FUNCTION_BLOCK Updater_1 IMPLEMENTS ITF_Updater
VAR CONSTANT
    PacketID  				: BYTE := 1;
    PacketVersion 			: BYTE := 1;
	PacketSize				: BYTE := 66;
END_VAR
VAR
	TempBuffer				: ARRAY [0..PacketSize - 1] OF BYTE;	

	ApplyOkCount            : UDINT;
    ApplyLengthErrorCount   : UDINT;
    ApplyBufferTooSmall     : UDINT;
END_VAR

METHOD GetTypeID : BYTE
GetTypeID := PacketID;
END_METHOD

METHOD GetVersion : BYTE
GetVersion := PacketVersion;
END_METHOD

METHOD TryApplyPayload : HRESULT
VAR_INPUT
	PacketAddress	: PVOID;
	PacketLength	: UINT;
	EspHost			: ITF_EspHost;
END_VAR
VAR
    BufferAddress : PVOID;
    BufferSize    : UDINT;
END_VAR
TryApplyPayload := S_PENDING;

IF PacketLength <> PacketSize THEN
	
    ApplyLengthErrorCount := ApplyLengthErrorCount + 1;
	
	TryApplyPayload := -1;
	
	RETURN;
	
END_IF

IF NOT EspHost.GetDataBuffer(BufferAddress, BufferSize) THEN
	
	TryApplyPayload := -2;

    RETURN;
	
END_IF

IF PacketLength > BufferSize THEN
	
    ApplyBufferTooSmall := ApplyBufferTooSmall + 1;
	
    TryApplyPayload := -3;
    
	RETURN;

END_IF



MEMCPY(BufferAddress, PacketAddress, PacketLength);

ApplyOkCount := ApplyOkCount + 1;

TryApplyPayload := S_OK;          // success

RETURN;
END_METHOD

METHOD TryGetContents : HRESULT
VAR_INPUT
	Host	: ITF_EspHost;
	Content	: REFERENCE TO STRING(1024);
END_VAR
VAR
    BufferAddress 	: PVOID;
    BufferSize   	: UDINT;
	td9 			: ULINT;
END_VAR
TryGetContents := S_PENDING;

Content := '{"Error" : "No_Data_Available"}';

IF NOT Host.GetDataBuffer(BufferAddress, BufferSize) THEN

	TryGetContents := -1;	

    RETURN;
	
END_IF

IF MEMCPY(ADR(TempBuffer), BufferAddress, BufferSize) <= 0 THEN
	
	TryGetContents := -2;
	
	RETURN;

END_IF

Content := '';

Content := CONCAT(Content, '{"Test_Data_1" : ');
Content := CONCAT(Content, TO_STRING(TempBuffer[48]));
Content := CONCAT(Content, ', "Test_Data_2" : ');
Content := CONCAT(Content, TO_STRING(TempBuffer[49]));
Content := CONCAT(Content, ', "Test_Data_3" : ');
Content := CONCAT(Content, TO_STRING(TempBuffer[50]));
Content := CONCAT(Content, ', "Test_Data_4" : ');
Content := CONCAT(Content, TO_STRING(TempBuffer[51]));
Content := CONCAT(Content, ', "Test_Data_5" : ');
Content := CONCAT(Content, TO_STRING(TempBuffer[52]));
Content := CONCAT(Content, ', "Test_Data_6" : ');
Content := CONCAT(Content, TO_STRING(TempBuffer[53]));
Content := CONCAT(Content, ', "Test_Data_7" : ');
Content := CONCAT(Content, TO_STRING(TempBuffer[54]));
Content := CONCAT(Content, ', "Test_Data_8" : ');
Content := CONCAT(Content, TO_STRING(TempBuffer[55]));

td9 := (TempBuffer[56]);
td9 := SHL(td9, 8) OR (TempBuffer[57]);
td9 := SHL(td9, 8) OR (TempBuffer[58]);
td9 := SHL(td9, 8) OR (TempBuffer[59]);
td9 := SHL(td9, 8) OR (TempBuffer[60]);
td9 := SHL(td9, 8) OR (TempBuffer[61]);
td9 := SHL(td9, 8) OR (TempBuffer[62]);
td9 := SHL(td9, 8) OR (TempBuffer[63]);

Content := CONCAT(Content, ', "Test_Data_9" : ');
Content := CONCAT(Content, TO_STRING(td9));
Content := CONCAT(Content, '}');

TryGetContents := S_OK;

RETURN;
END_METHOD

{warning 'Add method implementation '}
METHOD TrySendInstruction : HRESULT
END_METHOD

END_FUNCTION_BLOCK

(* stored: Version 1.1.0.1
   POU Updater_1: Id {bd79bccd-023d-4c74-aa4d-f04321d65ae1}, SpecialFunc None
   Folder ITF_Updater: Id {dff51703-c49a-4fcb-b6fc-3de4a0a9c731}
   Method GetTypeID: Id {509ff72a-6577-43fb-95d5-49f461ecdabc}
   Method GetVersion: Id {3d91a00b-8b56-4dc7-bcda-df8b40561b35}
   Method TryApplyPayload: Id {ddc6e7b4-b65e-41a4-8326-cf3a5a73d169}
   Method TryGetContents: Id {f327ca8a-76cb-444c-8ebc-989c3d6d118d}
   Method TrySendInstruction: Id {2fb1adb3-7a93-42a3-89c8-dde3be6bb528} *)
